FUNCTION_BLOCK FB_AxisReadParams
VAR_INPUT
	bExecute: BOOL;
	bReset: BOOL;
END_VAR
VAR_OUTPUT
	stConfig: ST_AxisParams;
	bValid: BOOL;
	bBusy: BOOL;
	bError: BOOL;
	iErrorID: UDINT;
END_VAR
VAR_IN_OUT
	Axis: AXIS_REF;
END_VAR
VAR
	fbNCRead: FB_AxisReadNC;
	fbCoERead: FB_AxisReadCoE;
END_VAR

fbNCRead(bExecute:=bExecute,
	bReset:=bReset,
	stConfig:=stConfig,
	Axis:=Axis,
	bValid=>bValid,
	bBusy=>bBusy,
	bError=>bError,
	iErrorID=>iErrorID);

END_FUNCTION_BLOCK

(* stored: Version 1.1.0.1, ProductVersion 3.1.4020.12
   POU FB_AxisReadParams: Id {e92502d6-67ee-4fa0-a7de-4596fc050760}, SpecialFunc None *)
